(* IEC 61131-3 sources: actions-test/src, 1 file *)

(* ---- library.st ---- *)
NAMESPACE MyLibrary

    CLASS PUBLIC MyClass
        VAR PUBLIC

        END_VAR

        VAR PRIVATE

        END_VAR

        METHOD PUBLIC DescriptiveMethodName : BOOL
            DescriptiveMethodName := FALSE;
        END_METHOD
    END_CLASS

END_NAMESPACE
